# EPICS substitutions: OceanopticsApp/Db/user.substitutions
# SPDX-FileCopyrightText: 2006 Argonne National Laboratory
#
# SPDX-License-Identifier: EPICS

# Example substitutions file

file "db/circle.db" {
    { user = "chem_epics" }
}

file "db/dbExample1.db" {
    { user = "chem_epics" }
}

file db/dbExample2.db {
    pattern { user, no, scan }
        { "chem_epics", 1, "1 second" }
        { "chem_epics", 2, "2 second" }
        { "chem_epics", 3, "5 second" }
}
